{attribute 'linkalways'} 
{attribute 'no_explicit_call' := 'This FB is a CLASS and must be accessed using methods or properties'}
{attribute 'enable_dynamic_creation'}
FUNCTION_BLOCK ABSTRACT InterfaceDatatypeBase EXTENDS DatatypeBase IMPLEMENTS I_InterfaceDatatype
VAR
END_VAR

PROPERTY PUBLIC ABSTRACT Identifier : T_MAXSTRING
GET
END_GET
END_PROPERTY

PROPERTY PUBLIC IsUserDefined : BOOL
GET
IsUserDefined := FALSE;
END_GET
END_PROPERTY

METHOD PROTECTED OnSerializeTypeWith
VAR_INPUT
	Serializer : I_Serializer;
END_VAR
SUPER^.OnSerializeTypeWith(Serializer);
Serializer.AddKeyString('identifier',Identifier);
END_METHOD

METHOD PUBLIC ABSTRACT TryCopyContentFrom : BOOL
VAR_INPUT
	Source : I_InterfaceDatatype;
END_VAR
END_METHOD

METHOD PUBLIC TryCopyFrom : BOOL
VAR_INPUT
	Source : I_Datatype;
END_VAR
VAR
	sourceAsInterface : I_InterfaceDatatype;
END_VAR
IF NOT Source.TryResolveAsInterfaceDatatype(sourceAsInterface) THEN
	RETURN;
END_IF

IF sourceAsInterface.Identifier <> Identifier THEN
	RETURN;
END_IF

TryCopyFrom := SUPER^.TryCopyFrom(Source);
END_METHOD

METHOD PUBLIC TryResolveAsInterfaceDatatype : BOOL
VAR_INPUT
	Destination : REFERENCE TO I_InterfaceDatatype;
END_VAR
Destination := THIS^;
TryResolveAsInterfaceDatatype := TRUE;
END_METHOD

PROPERTY PUBLIC TypeName : T_MAXSTRING
GET
TypeName := 'INTERFACE';
END_GET
END_PROPERTY

END_FUNCTION_BLOCK

(* stored: Version 1.1.0.1, ProductVersion 3.1.4026.18
   POU InterfaceDatatypeBase: Id {e46856b8-787d-4373-948a-d9f8155b7484}, SpecialFunc None
   Folder Protected: Id {9b22b654-1da4-40aa-b14a-7c7c6088cf5e}
   Property Identifier: Id {e8fe1895-9f44-4ce4-b3de-4d156c5d4ad7}
   Get Get: Id {9a8e2f09-755b-4b24-8e18-65db8adbd73e}
   Property IsUserDefined: Id {790f0c75-292a-4239-9b3a-596f0735bcde}
   Get Get: Id {453bbc2c-3677-443e-8223-ec5b4a40bb41}
   Method OnSerializeTypeWith: Id {f4c92b18-c542-47e9-875b-196b6bf83ecb}
   Method TryCopyContentFrom: Id {2fb0b68b-0476-077e-1133-20e124f86f6b}
   Method TryCopyFrom: Id {a0a4bb8e-cd4f-4087-b39c-d977c7f809fa}
   Method TryResolveAsInterfaceDatatype: Id {fbe47ae7-86c1-436d-981d-e0ad765eb393}
   Property TypeName: Id {123773f6-6f20-4d1f-9838-b3a78f7e3bf2}
   Get Get: Id {1ddd989a-5048-44e0-99ed-d7e6c17d1779} *)
